// TIA Portal project "IOT2050_OPCUA_CompleteProject" (V16)

(* hardware
DEVICE "ET 200SP station_1"  ET 200SP-Station
   slot 0: "Rack_0"  Rack  6ES5 710-8MAx1
   slot 1: "PLC_1"  CPU 1512SP F-1 PN  6ES7 512-1SK01-0AB0  V2.5
   slot 2: "Server module_1"  Server module  6ES7 193-6PA00-0AA0  V1.1
      slot 1: "Server module_1"  Server module
   slot 127: "BA 2xRJ45"  BA 2xRJ45  6ES7 193-6AR00-0AA0  V0.0
      slot 32769: "Port_1"  6ES7 193-6AR00-0AA0
      slot 32770: "Port_2"  6ES7 193-6AR00-0AA0
*)

// ===== PLC "PLC_1"  CPU 1512SP F-1 PN =====

DATA_BLOCK "Temperature Control_DB"   // DB2
{ S7_Optimized_Access := 'TRUE' }
VERSION : 0.1
// stored: InstanceOfName Temperature Control
"Temperature Control"
BEGIN
END_DATA_BLOCK

// folder: 02_OPCUA

DATA_BLOCK "OPC_UA_DB"   // DB1
{ S7_Optimized_Access := 'TRUE' }
VERSION : 0.1
   VAR
      TO_IOT2050 : Struct   // Read Access for IOT2050
         heaterOutput : Real := 0.0;   // 0 to 100% output for heater
         coolerOutput : Real := 0.0;   // 0 to 100% output for cooler
         actualTemperature : Real := 0.0;   // actual temperature reading n °C
         heaterStatus : Bool := false;   // 0 = Heater is OFF; 1 = Heater is ON
         coolerStatus : Bool := false;   // 0 = Cooler is OFF; 1 = Cooler is ON
      END_STRUCT;
      FROM_IOT2050 : Struct   // Write Access for IOT2050
         tempSetpoint : Real := 0.0;   // temperature setpoint in °C
      END_STRUCT;
   END_VAR
BEGIN
END_DATA_BLOCK

// folder: (top level)

ORGANIZATION_BLOCK "Main"   // OB1, LAD, ProgramCycle
TITLE = "Main Program Sweep (Cycle)"
{ S7_Optimized_Access := 'TRUE' }
VERSION : 0.1
   VAR_INPUT
      Initial_Call : Bool;   // Initial call of this OB
      Remanence : Bool;   // =True, if remanent data are available
   END_VAR
BEGIN

REGION Network 1
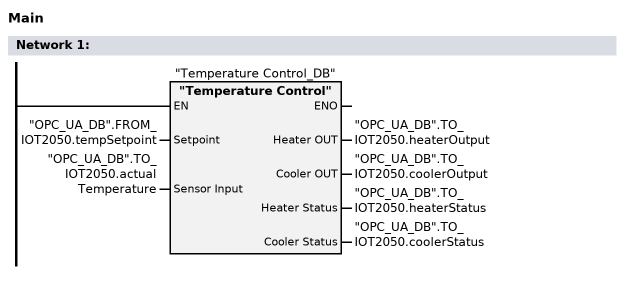
   RUNG wire#powerrail
      "Temperature Control_DB"(Setpoint := "OPC_UA_DB".FROM_IOT2050.tempSetpoint, "Sensor Input" := "OPC_UA_DB".TO_IOT2050.actualTemperature, "Heater OUT" => "OPC_UA_DB".TO_IOT2050.heaterOutput, "Cooler OUT" => "OPC_UA_DB".TO_IOT2050.coolerOutput, "Heater Status" => "OPC_UA_DB".TO_IOT2050.heaterStatus, "Cooler Status" => "OPC_UA_DB".TO_IOT2050.coolerStatus)
   END_RUNG
   // the same network as SCL:
   "Temperature Control_DB"(Setpoint := "OPC_UA_DB".FROM_IOT2050.tempSetpoint,   // "Temperature Control"
                           "Sensor Input" := "OPC_UA_DB".TO_IOT2050.actualTemperature,
                           "Heater OUT" => "OPC_UA_DB".TO_IOT2050.heaterOutput,
                           "Cooler OUT" => "OPC_UA_DB".TO_IOT2050.coolerOutput,
                           "Heater Status" => "OPC_UA_DB".TO_IOT2050.heaterStatus,
                           "Cooler Status" => "OPC_UA_DB".TO_IOT2050.coolerStatus);
END_REGION
END_ORGANIZATION_BLOCK

// folder: 02_OPCUA

FUNCTION_BLOCK "Temperature Control"   // FB1, LAD
{ S7_Optimized_Access := 'TRUE' }
VERSION : 0.1
   VAR_INPUT
      Setpoint : Real := 0.0;   // temperature setpoint in °C
   END_VAR
   VAR_OUTPUT
      "Heater OUT" : Real := 0.0;   // 0 to 100% output for heater
      "Cooler OUT" : Real := 0.0;   // 0 to 100% output for cooler
      "Heater Status" : Bool := false;   // 0 = Heater is OFF; 1 = Heater is ON
      "Cooler Status" : Bool := false;   // 0 = Cooler is OFF; 1 = Cooler is ON
   END_VAR
   VAR_IN_OUT
      "Sensor Input" : Real := 0.0;   // actual temperature reading n °C
   END_VAR
BEGIN

REGION Network 1: Closed Loop PID Temperature Control
   // By default its in Automatic mode
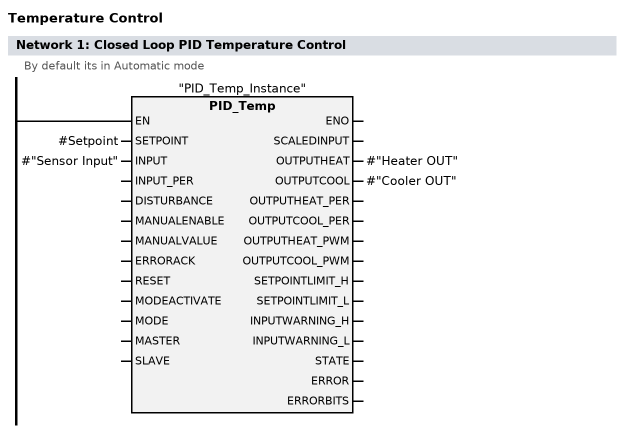
   "PID_Temp_Instance"(Setpoint := #Setpoint,   // PID_Temp
                       Input := #"Sensor Input",
                       OutputHeat => #"Heater OUT",
                       OutputCool => #"Cooler OUT");
END_REGION

REGION Network 2 (SCL): Simulate thermocouple sensor reading
   IF #"Heater OUT" > 0 THEN // increase temperature by adding heat
       #"Sensor Input" := #"Sensor Input" + (#"Heater OUT" / 10000);

   ELSIF #"Cooler OUT" > 0 THEN // decrease temperature by removing heat
       #"Sensor Input" := #"Sensor Input" - (#"Cooler OUT" / 10000);

   ELSE // do nothing
       ;
   END_IF;
END_REGION

REGION Network 3 (SCL): Converts % output of a heater or cooler to Boolean (ON/OFF) for Status
   IF #"Heater OUT" > 0 THEN
       #"Heater Status" := TRUE;
   ELSE
       #"Heater Status" := FALSE;
   END_IF;

   IF #"Cooler OUT" > 0 THEN
       #"Cooler Status" := TRUE;
   ELSE
       #"Cooler Status" := FALSE;
   END_IF;
END_REGION
END_FUNCTION_BLOCK